Universal Robots PolyScope program: setup.urp

Program setup (installation=default directory=/programs/Neuer Ordner createdIn=5.9.5.1031259 lastSavedIn=5.9.5.1031259 robotSerialNumber=20215000780)
Calibrated DH parameters: a=[-0.000076, -0.457222, -0.535711, -0.000049, -0.000015, 0]; d=[0.180847, -379.989416, 320.368416, 59.795924, 0.120055, 0.115601]; alpha=[1.570333, -0.001071, -0.003328, 1.572059, -1.570368, 0]; deltaTheta=[0, 0.727455, -0.372784, -0.354674, 0, 0]
Robot Program (runOnlyOnce=false)
  Placeholder
